TYPE ST_IoTDataHMI :
STRUCT
	Label 				: STRING;
	Varname				: eDataMappingVarNames;
	Unit				: STRING(20);
	LogType 			: eLogType; 
	LogInterval 		: eUpdate;
	b_IOTWriteAllowed	: BOOL;
END_STRUCT
END_TYPE

(* stored: Version 1.1.0.1, ProductVersion 3.1.4026.18
   DUT ST_IoTDataHMI: Id {752467d9-2fde-4476-812e-ef4b395f095e} *)
